// TIA Portal V20 export
// export: Created 2025-12-01T14:57:12.7770416Z, ExportSetting None, DisplayName Totally Integrated Automation Portal, DisplayVersion V20 Update 3, DisplayName TIA Portal Openness, DisplayVersion V20 Update 3, DisplayName TIA Portal Version Control Interface, DisplayVersion V20 Update 3, DisplayName STEP 7 Professional, DisplayVersion V20 Update 3, DisplayName STEP 7 Safety, DisplayVersion V20 Update 2, DisplayName WinCC Basic/Comfort/Advanced, DisplayVersion V20 Update 3, DisplayName WinCC Professional, DisplayVersion V20 Update 3, DisplayName WinCC Unified, DisplayVersion V20 Update 3
FUNCTION "FC755_EventosApilaDesApila" : Void   // FC755, STL
TITLE = Emision de los Eventos del Apilador-DesApialdor
{ S7_Optimized_Access := 'FALSE' }
AUTHOR : TRACKING
NAME : 20141014
VERSION : 4.0
// stored: AutoNumber false
   VAR_INPUT
      NumMaquina : UInt;   // Numero de Maquina
      EstadoMaquina : "EstadoZona";   // Estado de la Maquina
      EstadoVIMaquina : "EstadoMaquina";   // Estado del VI de la Maquina
      ApiladorVacio : Bool;   // Apilador esta Vacio
      ApiladorSemiLleno : Bool;   // Apilador esta SemiLleno
      ApiladorLleno : Bool;   // Apilador esta LLeno
      MesaDeJDT02 : Bool;
   END_VAR
   VAR_TEMP
      EstadoActual : UInt;
      P_EmiEventos : DWord;
      DBEventos : Word;
      NumBytes : UInt;
      OffsetInicial : UInt;
      OffsetFinal : UInt;
      Conversion : DWord;
      Convertir : UInt;
      Valor : UDInt;
      NumDBEventos : UInt;
      MaxBytes : UInt;
   END_VAR
BEGIN

NETWORK
TITLE = Inicializaciones
///////////////////////////////////////////////////////////////////////////////
/// Inicio --> Pertenece al JDT 02

      L     "JDT1_NDB_EventosEmi";
      T     #DBEventos;
      T     #NumDBEventos;
      L     "JDT1_MaxBytes";
      T     #MaxBytes;

      AN    #MesaDeJDT02;
      JC    NoJdT02;

      L     "JDT2_NDB_EventosEmi";
      T     #DBEventos;
      T     #NumDBEventos;
      L     "JDT2_MaxBytes";
      T     #MaxBytes;

NoJdT02:NOP   0;

/// Final --> Pertenece al JDT 02
///////////////////////////////////////////////////////////////////////////////




NETWORK
TITLE = Mirar si se pueden generar eventos
// - Inicializo el Numero de Bytes y el puntero del DB de Eventos Generados
// - Calcula el Tamaño de bytes que hay en el DB de Eventos Genardos
// - Comprobamos si hay sitio para Eventos
///////////////////////////////////////////////////////////////////////////////
/// Inicializo el Numero de Bytes y el puntero del DB Eventos Generados

      L     0;
      T     #NumBytes;  // Inicializo el numero de Bytes
      LAR2;  // Inicializo el puntero de Eventos Generados

///////////////////////////////////////////////////////////////////////////////
/// Calcula el tamaño de bytes que hay en el DB Eventos Generados

      OPN   DB [#DBEventos];

Inicio_BusquedaFinalEventos:NOP   0;
      L     DBB [AR2, P#0.0];
      L     0;
      ==I;
      JC    Final_BusquedaFinalEventos;  // Buscamos el final del DB = 0

      +AR2  P#1.0;
      JU    Inicio_BusquedaFinalEventos;

Final_BusquedaFinalEventos:NOP   0;
      TAR2;  // Guardo el puntero
      T     #P_EmiEventos;  // Sacamos el NumBytes Escritos
      SRD   3;
      T     #NumBytes;

// -----------------------------------------------------------------------------------------------
// Comprobamos si hay sitio para mas Eventos

      L     #NumBytes;  // Miramos si hay sitio
      L     #MaxBytes;  // Max. que se pueden emitir, parametro
      >I;
      JC    Final;  // No se pueden generar más eventos


NETWORK
TITLE = Distribucion
///////////////////////////////////////////////////////////////////////////////
// --- Distribucion  del Estado de Trabajo del Apilador

      L     0;
      T     #EstadoActual;

// ---------- Mirar si esta Vacio el Apilador

      A     #ApiladorVacio;
      AN    #ApiladorSemiLleno;
      AN    #ApiladorLleno;
      JCN   _ST1;  // No Esta Vacio ?

      L     1000;  // Esta Vacio
      T     #EstadoActual;
      JU    _STF;


// ---------- Mirar si esta Semi-Lleno el Apilador

_ST1: AN    #ApiladorVacio;
      A     #ApiladorSemiLleno;
      AN    #ApiladorLleno;
      JCN   _ST2;  // No Esta Semi-Lleno ?

      L     1001;  // Esta Semi-Lleno
      T     #EstadoActual;
      JU    _STF;


// ---------- Mirar si esta Lleno el Apilador

_ST2: AN    #ApiladorVacio;
      AN    #ApiladorSemiLleno;
      A     #ApiladorLleno;
      JCN   _ST3;  // No Esta Lleno ?

      L     1002;  // Esta Lleno
      T     #EstadoActual;
      JU    _STF;


// ---------- No se sabe como esta el apilador

_ST3: L     0;  // No se Sabe el Status de Trabajo
      T     "DB832_Maquinas".Maquinas[#NumMaquina].MemoriaEstado;

      JU    ST_F;


///////////////////////////////////////////////////////////////////////////////
// ---------- Mirar si hay que Emitir el Evento

_STF: L     "DB832_Maquinas".Maquinas[#NumMaquina].Operacion;
      L     5000;  // Peticion de Status del Apilador
      <>I;
      JC    ST_F;

      L     #EstadoActual;
      L     0;  // Existe Status del Apilador
      ==I;
      JC    ST_F;

      JU    EmisionDelEvento;


///////////////////////////////////////////////////////////////////////////////
// --- Fin del Estado de Trabajo del Apilador

ST_F: JU    Final;



NETWORK
TITLE = Emision del Evento
///////////////////////////////////////////////////////////////////////////////
// --- Formateo del Evento DIDA - Estado del Apilador - DesApilador

EmisionDelEvento:NOP   0;
      L     #P_EmiEventos;
      LAR2;  // Puntero al DB de Eventos Generados

      TAR2;  // Mirar si es el primer evento de la lista
      L     0;
      ==I;
      JC    NoEsInicio_ListaDeEventos;  // Es el primero

      OPN   DB [#DBEventos];
      L     ',';  // Separador entre eventos ','
      T     DBB [AR2, P#0.0];
      +AR2  P#1.0;

NoEsInicio_ListaDeEventos:NOP   0;
      OPN   DB [#DBEventos];  // DB de Eventos Generados (A Emitir)
      L     '{';  // Inicio de Evento '{'
      T     DBB [AR2, P#0.0];
      +AR2  P#1.0;


///////////////////////////////////////////////////////////////////////////////
// --- Cuerpo del Evento

      L     'DIDA';  // Evento 'DIDA'
      T     DBD [AR2, P#0.0];
      +AR2  P#4.0;

      OPN   DB [#DBEventos];
      L     '[';  // Evento - Atributo Tipo '[TIPO]'
      T     DBB [AR2, P#0.0];
      L     'TIPO';
      T     DBD [AR2, P#1.0];
      L     ']';
      T     DBB [AR2, P#5.0];
      +AR2  P#6.0;

      L     "DB850_DefinicionMesas".Mesa[#NumMaquina].ConfigMesa.TipoMaquina;
      T     #Convertir;

      CALL  "FC895_Obtener_EtiquetaDeValor"
      ( ValorEvento    := #Convertir,
        EtiquetaEvento := #Conversion
      );

      OPN   DB [#DBEventos];
      L     #Conversion;
      T     DBD [AR2, P#0.0];
      +AR2  P#4.0;


      L     '[';  // Evento - Atributo Numero de Dispositivo '[NUME]'
      T     DBB [AR2, P#0.0];
      L     'NUME';
      T     DBD [AR2, P#1.0];
      L     ']';
      T     DBB [AR2, P#5.0];
      +AR2  P#6.0;

      L     "CTE_OffsetMesa";
      L     #NumMaquina;  // Numero de Maquina
      +I;
      T     #Valor;

// --- Convertir Valor a ASCII - Numero de Maquina
      TAR2;
      SRD   3;
      T     #OffsetInicial;  // Miro que offset tiene la String

      CALL  "FC893_Obtener_StringDelAtributo"
      ( DB_String := #NumDBEventos,
        OffsetIni := #OffsetInicial,
        Valor     := #Valor,
        OffsetFin := #OffsetFinal
      );  // Llamo a ObtenerStrinAtributo

      L     #OffsetFinal;
      SLD   3;
      LAR2;  // Recupero que offset tiene la String

// --- Ya esta convertido el Valor a ASCII

      OPN   DB [#DBEventos];
      L     '[';  // Evento - Atributo Numero de Dispositivo '[FULL]'
      T     DBB [AR2, P#0.0];
      L     'FULL';
      T     DBD [AR2, P#1.0];
      L     ']';
      T     DBB [AR2, P#5.0];
      +AR2  P#6.0;

      L     #EstadoActual;  // Estado Actual del Apilador
      T     #Convertir;

      CALL  "FC895_Obtener_EtiquetaDeValor"
      ( ValorEvento    := #Convertir,
        EtiquetaEvento := #Conversion
      );

      OPN   DB [#DBEventos];
      L     #Conversion;
      T     DBD [AR2, P#0.0];
      +AR2  P#4.0;


///////////////////////////////////////////////////////////////////////////////
// Final del formateo del Evento

      OPN   DB [#DBEventos];  // DB de Eventos Generados (A Emitir)
      L     '}';  // Fin de Evento '}'
      T     DBB [AR2, P#0.0];
      +AR2  P#1.0;

///////////////////////////////////////////////////////////////////////////////
// Dar por formateado el Evento

      L     #EstadoActual;  // Lo doy por tratado
      T     "DB832_Maquinas".Maquinas[#NumMaquina].MemoriaEstado;
      L     0;
      T     "DB832_Maquinas".Maquinas[#NumMaquina].Operacion;

      JU    Final;  // Ya se ha generado el evento de la Maquina

// Fin del Formateo del Evento DIDA (Apilador)
///////////////////////////////////////////////////////////////////////////////
///////////////////////////////////////////////////////////////////////////////



NETWORK
TITLE = Fin de la Funcion
///////////////////////////////////////////////////////////////////////////////
//// -- Final de la Funcion
Final:NOP   0;



END_FUNCTION
